(* CODESYS project FU_wFindRight.xml

Project tree, tasks and I/O mapping:
  function FU_wFindRight [ST]
*)

// FU_wFindRight
//This function, returns the lenght of a string
// |**Version**|**Author**| **Date** |**Changes**
// | 1         | NSN      | 13-06-18 | Creation
FUNCTION FU_wFindRight : WORD
VAR_INPUT
	s1			:STRING(255);		//Input String1
	s2			:STRING(255);		//Input String2
END_VAR

FU_wFindRight	:=		FU_wFindRightBI(s1:=s1,s2:=s2);

END_FUNCTION
